# B&R Automation Studio project MpTempSample
Automation Studio 4.3.7.46 SP; technology packages: mappControl 5.2.0

## Configuration Config1

CPU X20CP1301, AutomationRuntime G4.34, Build 4.1.2

### Task classes (Cpu.sw)
```
Cyclic#4:
  Program <- Program.prg
Binaries: udbdef, arsvcreg, TCData, arconfig, User, sysconf, Role, Config, iomap, asfw, ashwac, ashwd, Config_1
Libraries: AsArProf, runtime, astime, asieccon, fileio, MpTemp, MTBasics, MpBase, brsystem, MTTypes, sys_lib, standard
```

### Hardware
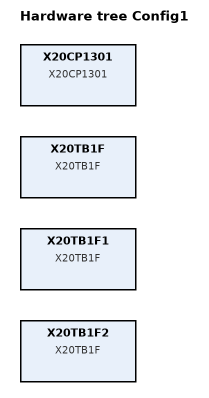
```
X20CP1301 : X20CP1301 v1.6.1.0  [X1 -> X1.SL; X2 -> X2.SL; X3 -> X3.SL]
  Module X1 (Type=X1, Virtual=true, Version=1.6.1.0)
    Connection (Connector=SS1, TargetModule=X20TB1F, TargetConnector=SS)
    Connection (Connector=SL, TargetModule=X20CP1301, TargetConnector=X1)
  Module X2 (Type=X2, Virtual=true, Version=1.6.1.0)
    Connection (Connector=SS1, TargetModule=X20TB1F1, TargetConnector=SS)
    Connection (Connector=SL, TargetModule=X20CP1301, TargetConnector=X2)
  Module X3 (Type=X3, Virtual=true, Version=1.6.1.0)
    Connection (Connector=SS1, TargetModule=X20TB1F2, TargetConnector=SS)
    Connection (Connector=SL, TargetModule=X20CP1301, TargetConnector=X3)
  Connector IF2:
    ActivateDevice = 1
    Mode = Manual
    InternetAddress = 192.168.0.7
    SubnetMask = 255.255.255.0
    InaNodeNumber = 7
    Vnc1
    VncKeyMappingFile1 = VC\PS2-Keyboard.dis
    VncRefreshRate1 = 300
  ConfigurationID = Heat_400252100_Config2
X20TB1F : X20TB1F v1.0.0.0
X20TB1F1 : X20TB1F v1.0.0.0
X20TB1F2 : X20TB1F v1.0.0.0
```

### Config.tempcontroller - X20CP1301/mappControl/Config.tempcontroller
```
Element gTempController01 (Type=tempcontroller)
  TempController:
    MaxHeatOutput = 100
    PWMParameters:
      Heat:
        Period = 2.0
Element gTempController02 (Type=tempcontroller)
  TempController:
    PWMParameters:
      Heat:
        Period = 2.0
Element gTempController03 (Type=tempcontroller)
  TempController:
    PWMParameters:
      Heat:
        Period = 2.0
Element gTempController04 (Type=tempcontroller)
  TempController:
    PWMParameters:
      Heat:
        Period = 2.0
Element gTempController05 (Type=tempcontroller)
  TempController:
    PWMParameters:
      Heat:
        Period = 2.0
Element gTempController06 (Type=tempcontroller)
  TempController:
    PWMParameters:
      Heat:
        Period = 2.0
Element gTempController07 (Type=tempcontroller)
  TempController:
    PWMParameters:
      Heat:
        Period = 2.0
Element gTempController08 (Type=tempcontroller)
  TempController:
    PWMParameters:
      Heat:
        Period = 2.0
Element gTempController09 (Type=tempcontroller)
  TempController:
    PWMParameters:
      Heat:
        Period = 2.0
Element gTempController10 (Type=tempcontroller)
  TempController:
    PWMParameters:
      Heat:
        Period = 2.0
```

### Config_1.tempgroup - X20CP1301/mappControl/Config_1.tempgroup
```
Element gTempGroup (Type=tempgroup)
  Linking:
    Subnodes:
      Zone[0] = gTempController01
      Zone[1] = gTempController02
      Zone[2] = gTempController03
      Zone[3] = gTempController04
      Zone[4] = gTempController05
      Zone[5] = gTempController06
      Zone[6] = gTempController07
      Zone[7] = gTempController08
      Zone[8] = gTempController09
      Zone[9] = gTempController10
  TempGroup:
    EnableLoadBalancing = FALSE
```

## Logical view

Binary libraries used (declarations not repeated): operator, runtime, astime, AsIecCon, MTTypes, sys_lib, brsystem, AsArProf, MpTemp 5.02.0, MTBasics 5.02.0, MpBase 5.02.0, standard


### Program Logical/Program (IEC)

#### Cyclic.st - Cyclic code
```iecst
PROGRAM _CYCLIC

  (* -------------------------------------------------------------------
	state machine
   ------------------------------------------------------------------- *)
	CASE step OF
		0:
		IF start = TRUE THEN
			step := 1;
		END_IF

		1: (* set step = 1 to start tuning, done after about 1300 seconds *)
		IF TempGroup.Active AND allTempControllerActive THEN

			fubGetTime(enable := TRUE);
			IF fubGetTime.status = 0 THEN
				startTime := fubGetTime.DT1;
				step := 10;
			END_IF
		END_IF

		10:
		(* TempController[0].Tune := TRUE ;*)
		TempGroup.Tune := TRUE;
		step := 20;

		20:
		fubGetTime(enable := TRUE);
		IF fubGetTime.status = 0 THEN
			endTime := fubGetTime.DT1;
			diffTime := DiffDT( endTime, startTime );  (* measure time used for tuning *)
		END_IF
		IF allTempControllerTuningDone THEN
			step := 30;
		END_IF

		30:
		IF allTempControllerInSetpoint THEN
			enableDisturbance := TRUE;
			tonWait( IN:= FALSE, PT:= T#100s );
			step := 40;
		END_IF

		40:
		tonWait( IN:= TRUE ); (* wait and test the quality of control with 'disturbances' *)
		IF tonWait.Q THEN
			enableDisturbance := FALSE;
			start := 0;
			step := 0;
		END_IF

	END_CASE

  (* -------------------------------------------------------------------
	temperature controller
   ------------------------------------------------------------------- *)

	(* collective signals  *)
	allTempControllerActive := TRUE;
	allTempControllerInSetpoint := TRUE;
	allTempControllerTuningDone := TRUE;
	tuningError := FALSE;

	(* run temperature controller *)
	FOR n:= 0 TO 9 DO
		TC ACCESS ADR(TempController[n]);

		CASE n OF
		0: TC.MpLink := ADR(gTempController01);
		1: TC.MpLink := ADR(gTempController02);
		2: TC.MpLink := ADR(gTempController03);
		3: TC.MpLink := ADR(gTempController04);
		4: TC.MpLink := ADR(gTempController05);
		5: TC.MpLink := ADR(gTempController06);
		6: TC.MpLink := ADR(gTempController07);
		7: TC.MpLink := ADR(gTempController08);
		8: TC.MpLink := ADR(gTempController09);
		9: TC.MpLink := ADR(gTempController10);
		END_CASE

		(* for profiler *)
		LogEvent_0(enable := 1, objIdent := 123 , userEvent := profUSER_EVENT_START , pAddData :=0 , addDataLen := 0);

		TC (
			Enable := TRUE,
			Parameters := ADR(Parameter),
			SetTemperature := SetTemperature,
			ActualTemperature := _MTBasicsPT2[n].Out + ambientTemperature
		);

		(* for profiler *)
		LogEvent_0(enable := 1, objIdent := 123 , userEvent := profUSER_EVENT_STOP , pAddData :=0 , addDataLen := 0);

		(* collective signals *)
		IF NOT(TC.Active) THEN
			allTempControllerActive := FALSE;
		END_IF
		IF TC.Info.Tuning.State <> mpTEMP_TUNING_STATE_IN_SETPOINT THEN
			allTempControllerInSetpoint := FALSE;
		END_IF
		IF TC.Info.Tuning.State = mpTEMP_TUNING_STATE_ERROR THEN
			tuningError := TRUE;
		END_IF
		IF TC.TuningDone = FALSE THEN
			allTempControllerTuningDone := FALSE;
		END_IF
	END_FOR

	(* run group *)
	TempGroup(
		MpLink := ADR(gTempGroup),
		Enable := TRUE,

		Parameters := ADR(GroupParameter),
	);

  (* -------------------------------------------------------------------
	run simulation model
   ------------------------------------------------------------------- *)
	FOR n:= 0 TO 9 DO
		_MTBasicsTimeDelay[n](
			Enable := TRUE,
			(* In := 80* TempController[n].HeatValue / 100.0 *)  (* analogue actuator *)
			In := 80 * BOOL_TO_REAL(TempController[n].Heat)	 (* digital actuator *)
		);

		_MTBasicsPT2[n](
			Enable := TRUE,
			In := _MTBasicsTimeDelay[n].Out + disturbance
		 );
	END_FOR

  (* -------------------------------------------------------------------
	simulate disturbance
   ------------------------------------------------------------------- *)
   	IF enableDisturbance THEN
		disturbanceCounter := disturbanceCounter + 1;
		IF disturbanceCounter > 50 AND disturbanceCounter <= 60 THEN
			disturbance := 20;
		ELSIF disturbanceCounter > 60 THEN
			disturbance := 0;
			disturbanceCounter := 0;
		END_IF
	END_IF

END_PROGRAM
```

#### Init.st - Init code
```iecst
PROGRAM _INIT

	Parameter.ToleranceBand.Lower := 20;
	Parameter.ToleranceBand.Upper := 20;

	SetTemperature := 122;
	ambientTemperature := 25.0;
	disturbance := 0;
	enableDisturbance := FALSE;

	(* simulation model *)
	FOR n:= 0 TO 9 DO
		_MTBasicsTimeDelay[n](
			Enable := FALSE,
			DelayTime := 2.0 + n,
		);

		_MTBasicsPT2[n](
			Enable := FALSE,
			Gain := 15,
			TimeConstant1 := 200 + 20 * n,
			TimeConstant2 := 150 - 10 * n,
		 );

	END_FOR

END_PROGRAM
```

#### Variables.var - Local variables
```iecst
VAR
	tonWait : TON;
	disturbanceCounter : UINT;
	start : BOOL;
	startTime : DATE_AND_TIME;
	endTime : DATE_AND_TIME;
	fubGetTime : DTGetTime;
	diffTime : UDINT;
	TempController : ARRAY[0..9] OF MpTempController;
	TempGroup : MpTempGroup;
	Parameter : MpTempControllerParType;
	GroupParameter : MpTempGroupParType;
	n : INT;
	TC : REFERENCE TO MpTempController;
	step : UINT;
	allTempControllerActive : BOOL;
	_MTBasicsPT2 : ARRAY[0..9] OF MTBasicsPT2;
	_MTBasicsTimeDelay : ARRAY[0..9] OF MTBasicsTimeDelay;
	allTempControllerInSetpoint : BOOL;
	tuningError : BOOL;
	LogEvent_0 : LogEvent;
	SetTemperature : REAL;
	ambientTemperature : REAL;
	allTempControllerTuningDone : BOOL;
	disturbance : REAL;
	enableDisturbance : BOOL;
END_VAR
```

Listed in the project but not available here: Logical/Global.typ, Logical/Global.var, Logical/Program/Exit.st, Logical/Program/Types.typ
